{attribute 'qualified_only'}
{attribute 'strict'}
TYPE E_PneumaticMode :
(   SINGLE_SOLENOID_PLC := 0,
    SINGLE_SOLENOID_MANUAL := 1,
    ERROR := 2,
    RESET := 3
):= SINGLE_SOLENOID_PLC;
END_TYPE

(* stored: Version 1.1.0.1, ProductVersion 3.1.4024.5
   DUT E_PneumaticMode: Id {767ff514-f7ef-4e71-a359-d55b64a86d25} *)
